{attribute  'hide'}
TYPE ST_Event :
STRUCT
	EventType:T_MaxString;
	sEventText:T_MaxString;
	timesatamp:T_MaxString;
END_STRUCT
END_TYPE

(* stored: Version 1.1.0.1, ProductVersion 3.1.4024.6
   DUT ST_Event: Id {f75da5c5-6b58-4875-b104-70781c8fe24f} *)
